Xinje XDPPro project, PLC1: XD5-48T6 (software 3.5.3 2018-11-19)

PROGRAM Ladder

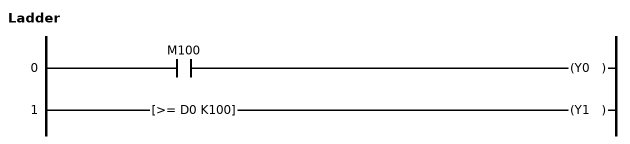
LD     M100
OUT    Y0
LD>=   D0 K100
OUT    Y1